DEVICE_TYPE DeviceType (* Device Type *)
  (* Standard: 61499-2 *)
  (* Version 0.2, 2003-12-05, JHC, Rockwell Automation, Renamed from NEWDEVICE. *)
  (* Version 0.1, 2002-11-05, JHC, Rockwell Automation, Corrected <DeviceFBNetwork> to <FBNetwork>. *)
  (* Version 0.0, 2000-05-27, JHC, Rockwell Automation *)
  (* Compiler header: package fb.rt.template; *)
  RESOURCE RES1 : ResourceType
  END_RESOURCE
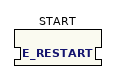
  FBS
    START : E_RESTART;
  END_FBS
END_DEVICE_TYPE
